Fanuc TP program (LS listing): MON_OP40ALM.LS

/PROG  MON_OP40ALM
/ATTR
OWNER		= MNEDITOR;
COMMENT		= "MONITOR ALARM";
PROG_SIZE	= 269;
CREATE		= DATE 20-02-06  TIME 06:36:06;
MODIFIED	= DATE 20-02-06  TIME 06:41:54;
FILE_NAME	= MON_OP10;
VERSION		= 0;
LINE_COUNT	= 3;
MEMORY_SIZE	= 645;
PROTECT		= READ_WRITE;
TCD:  STACK_SIZE	= 0,
      TASK_PRIORITY	= 50,
      TIME_SLICE	= 0,
      BUSY_LAMP_OFF	= 0,
      ABORT_REQUEST	= 0,
      PAUSE_REQUEST	= 0;
DEFAULT_GROUP	= *,*,*,*,*;
CONTROL_CODE	= 00000000 00000000;
/APPL

AUTO_SINGULARITY_HEADER;
  ENABLE_SINGULARITY_AVOIDANCE   : TRUE;
/MN
   1:  CALL MACH_MSG(15) ;
   2:  UALM[5] ;
   3:  MONITOR MON_OP40 ;
/POS
/END
